FUNCTION_BLOCK EHWCheckRange
VAR_INPUT
	rBarcodeReading : REAL; // current relative reading
	tsTrack : ST_Track_Segment_EHC; // current track segment
END_VAR
VAR_OUTPUT
	bResult : BOOL;
END_VAR
VAR
END_VAR

bResult := FALSE;

IF tsTrack.rStart < tsTrack.rEnd THEN
	IF rBarcodeReading >= tsTrack.rStart + 0.05 AND rBarcodeReading <= tsTrack.rEnd - 0.05 THEN
		bResult := TRUE;
	END_IF
ELSE
	IF rBarcodeReading <= tsTrack.rStart - 0.05 AND rBarcodeReading >= tsTrack.rEnd + 0.05 THEN
		bResult := TRUE;
	END_IF
END_IF

END_FUNCTION_BLOCK

(* stored: Version 1.1.0.1
   POU EHWCheckRange: Id {3685a3cf-2272-4ad8-a733-400df0e57c98}, SpecialFunc None *)
